FUNCTION_BLOCK IEEE1451_EVENT_SENSOR
  {SET_ATTRIBUTE(OpcUa, SERVICE)}
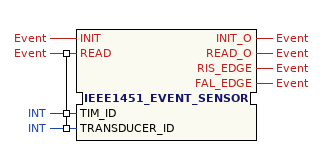
  EVENT_INPUT
    INIT; (* FB Initialization *)
    READ WITH TIM_ID, TRANSDUCER_ID; (* Read Sensor Request *)
  END_EVENT
  EVENT_OUTPUT
    INIT_O; (* Initialization Confirm *)
    READ_O; (* Read Request Confirm *)
    RIS_EDGE; (* Event Rising Edge *)
    FAL_EDGE; (* Event Falling Edge *)
  END_EVENT
  VAR_INPUT
    TIM_ID : INT; (* TIM Identification *)
    TRANSDUCER_ID : INT; (* Transducer Identification *)
  END_VAR
END_FUNCTION_BLOCK
